FUNCTION_BLOCK CompressorControl
VAR_INPUT
	MethodCall: BOOL;
	NotAus_Signal : BOOL;
	Destination : BOOL;
	LightSensor_01: BOOL;
	LightSensor_02: BOOL;
	TS_Endschalter_01: BOOL;
	TS_Endschalter_02: BOOL;
	EncoderStartPosition_01 : BOOL;
	EncoderStartPosition_02 : BOOL;
	EncoderStartPosition_03 : BOOL;
	EncoderStartPosition_04 : BOOL;
	EncoderStartPosition_05 : BOOL;
	EncoderStartPosition_06 : BOOL;
	EncoderTargetPosition_01 : BOOL;
	EncoderTargetPosition_02 : BOOL;
	EncoderTargetPosition_03 : BOOL;
	EncoderTargetPosition_04 : BOOL;
	EncoderTargetPosition_05 : BOOL;
	EncoderTargetPosition_06 : BOOL;	
	PowerOnDelay_Kompressor: TIME;
	PowerOnDelay_Ventil: TIME;
	AutomaticMode: BOOL;
END_VAR
VAR_OUTPUT
	Ansteuerung_Compressor : BOOL;
	Ansteuerung_Ventil : BOOL;
END_VAR
VAR
//FlipFlop
	RS_Vakuumkompressor: RS;
	RS_Vakuumventil: RS;
//Zeitverzögerung
	TON_Ansteuerung_Kompressor: TON;
	TON_Ansteuerung_Ventil: TON;
//Flanke	
	R_TRIG_MethodCall: R_TRIG;
END_VAR

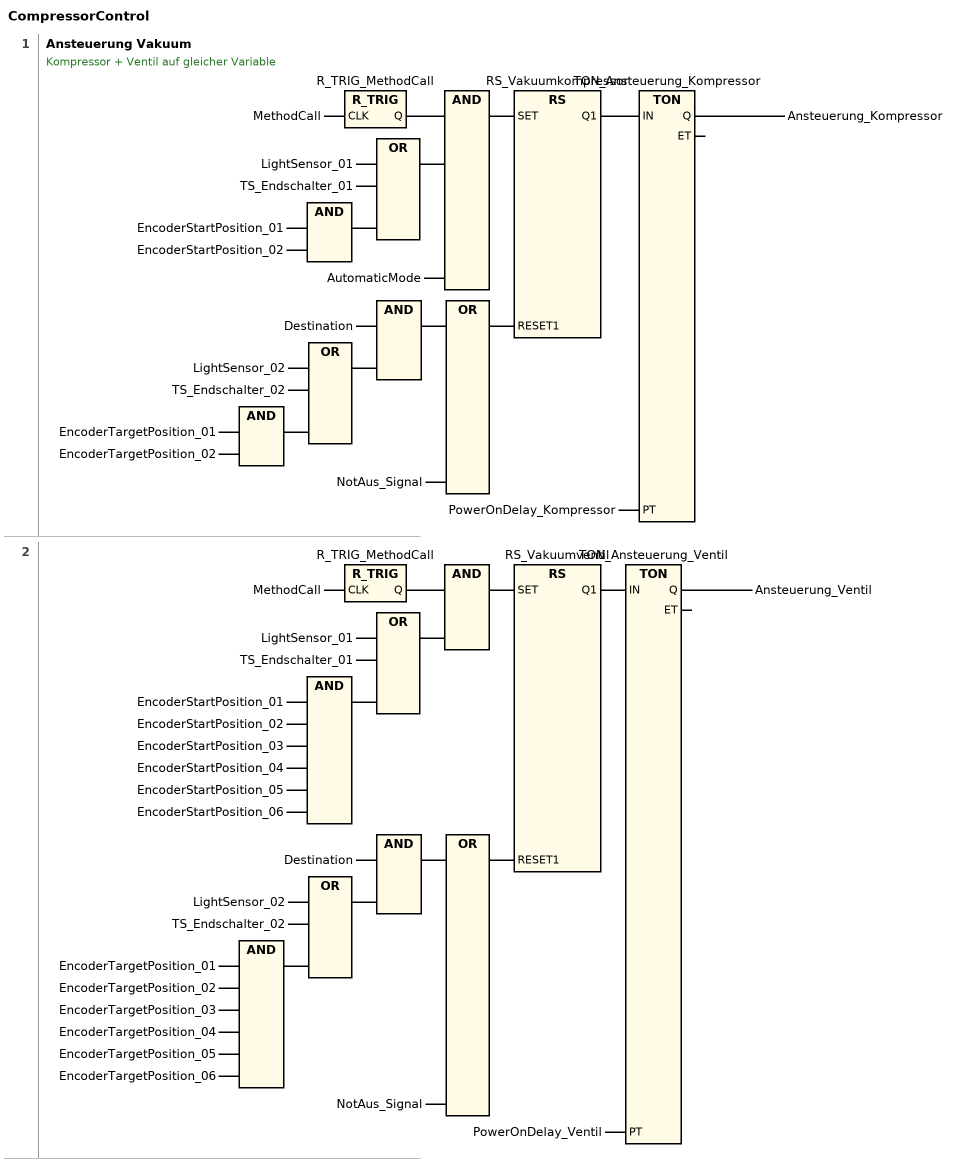
// NETWORK 1: Ansteuerung Vakuum
// Kompressor + Ventil auf gleicher Variable
R_TRIG_MethodCall(CLK := MethodCall); // R_TRIG
RS_Vakuumkompressor(SET := R_TRIG_MethodCall.Q AND (LightSensor_01 OR TS_Endschalter_01 OR EncoderStartPosition_01 AND EncoderStartPosition_02) AND AutomaticMode, RESET1 := Destination AND (LightSensor_02 OR TS_Endschalter_02 OR EncoderTargetPosition_01 AND EncoderTargetPosition_02) OR NotAus_Signal); // RS
TON_Ansteuerung_Kompressor(IN := RS_Vakuumkompressor.Q1, PT := PowerOnDelay_Kompressor); // TON
Ansteuerung_Kompressor := TON_Ansteuerung_Kompressor.Q;

// NETWORK 2
R_TRIG_MethodCall(CLK := MethodCall); // R_TRIG
RS_Vakuumventil(SET := R_TRIG_MethodCall.Q AND (LightSensor_01 OR TS_Endschalter_01 OR EncoderStartPosition_01 AND EncoderStartPosition_02 AND EncoderStartPosition_03 AND EncoderStartPosition_04 AND EncoderStartPosition_05 AND EncoderStartPosition_06), RESET1 := Destination AND (LightSensor_02 OR TS_Endschalter_02 OR EncoderTargetPosition_01 AND EncoderTargetPosition_02 AND EncoderTargetPosition_03 AND EncoderTargetPosition_04 AND EncoderTargetPosition_05 AND EncoderTargetPosition_06) OR NotAus_Signal); // RS
TON_Ansteuerung_Ventil(IN := RS_Vakuumventil.Q1, PT := PowerOnDelay_Ventil); // TON
Ansteuerung_Ventil := TON_Ansteuerung_Ventil.Q;

END_FUNCTION_BLOCK

(* stored: Version 1.1.0.1, ProductVersion 3.1.4024.15
   POU CompressorControl: Id {08453029-282a-4201-b8f6-3e5a26de7c2f}, SpecialFunc None *)
